SUBAPPLICATION Ventilsteuerung_Uebung_010b2 (* Toggle Flip-Flop mit IE SoftKey_F1 *)
  (* Standard: 61499-2 *)
  (* Version 1.0, 2023-10-23, franz *)
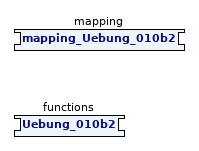
  SUBAPPS
    mapping : mapping_Uebung_010b2;
    functions : Uebung_010b2;
  END_SUBAPPS
END_SUBAPPLICATION
